(* IEC 61131-3 sources: DemoPumpStation/Testing, 3 files *)

(* ---- test_pdi_codec.st ---- *)
// @Test "PdiCodec decode with both command bits cleared"
// @data (control:=0, powerWord:=0, expectedStart:=0, expectedStop:=0, expectedPower:=0.0)
FUNCTION Test_PdiCodec_Decode_NoCommands : bool
VAR_INPUT
    control : word;
    powerWord : word;
    expectedStart : bool;
    expectedStop : bool;
    expectedPower : real;
END_VAR
VAR
    codec : PdiCodec;
    entry : PumpStationControl;
    words : array[0..1] of word;
    seg : Modbus.ModbusSegment;
END_VAR
    // Arrange
    words[0] := control;
    words[1] := powerWord;
    seg.attachReadable('mbs', Modbus.ModbusArea#holds, 0, ref(words));
    codec.init(0, seg);

    entry.startCmd := true;
    entry.stopCmd := true;
    entry.setpointPower := -999.0;

    // Act
    codec.decode(entry);

    // Assert
    Test_PdiCodec_Decode_NoCommands :=
        (entry.startCmd = expectedStart) and
        (entry.stopCmd = expectedStop) and
        (entry.setpointPower = expectedPower);
END_FUNCTION

// @Test "PdiCodec decode start command only"
// @data (control:=1, powerWord:=100, expectedStart:=1, expectedStop:=0, expectedPower:=100.0)
FUNCTION Test_PdiCodec_Decode_StartOnly : bool
VAR_INPUT
    control : word;
    powerWord : word;
    expectedStart : bool;
    expectedStop : bool;
    expectedPower : real;
END_VAR
VAR
    codec : PdiCodec;
    entry : PumpStationControl;
    words : array[0..1] of word;
    seg : Modbus.ModbusSegment;
END_VAR
    words[0] := control;
    words[1] := powerWord;

    seg.attachReadable('mbs', Modbus.ModbusArea#holds, 0, ref(words));
    codec.init(0, seg);

    entry.startCmd := false;
    entry.stopCmd := true;
    entry.setpointPower := -1.0;

    codec.decode(entry);

    Test_PdiCodec_Decode_StartOnly :=
        (entry.startCmd = expectedStart) and
        (entry.stopCmd = expectedStop) and
        (entry.setpointPower = expectedPower);
END_FUNCTION

// @Test "PdiCodec decode stop command only"
// @data (control:=2, powerWord:=250, expectedStart:=0, expectedStop:=1, expectedPower:=250.0)
FUNCTION Test_PdiCodec_Decode_StopOnly : bool
VAR_INPUT
    control : word;
    powerWord : word;
    expectedStart : bool;
    expectedStop : bool;
    expectedPower : real;
END_VAR
VAR
    codec : PdiCodec;
    entry : PumpStationControl;
    words : array[0..1] of word;
    seg : Modbus.ModbusSegment;
END_VAR
    words[0] := control;
    words[1] := powerWord;
    seg.attachReadable('mbs', Modbus.ModbusArea#holds, 0, ref(words));
    codec.init(0, seg);

    entry.startCmd := true;
    entry.stopCmd := false;
    entry.setpointPower := -1.0;

    codec.decode(entry);

    Test_PdiCodec_Decode_StopOnly :=
        (entry.startCmd = expectedStart) and
        (entry.stopCmd = expectedStop) and
        (entry.setpointPower = expectedPower);
END_FUNCTION

// @Test "PdiCodec decode both command bits set"
// @data (control:=3, powerWord:=500, expectedStart:=1, expectedStop:=1, expectedPower:=500.0)
FUNCTION Test_PdiCodec_Decode_BothCommands : bool
VAR_INPUT
    control : word;
    powerWord : word;
    expectedStart : bool;
    expectedStop : bool;
    expectedPower : real;
END_VAR
VAR
    codec : PdiCodec;
    entry : PumpStationControl;
    words : array[0..1] of word;
    seg : Modbus.ModbusSegment;
END_VAR
    words[0] := control;
    words[1] := powerWord;
    seg.attachReadable('mbs', Modbus.ModbusArea#holds, 0, ref(words));
    codec.init(0, seg);

    entry.startCmd := false;
    entry.stopCmd := false;
    entry.setpointPower := -1.0;

    codec.decode(entry);

    Test_PdiCodec_Decode_BothCommands :=
        (entry.startCmd = expectedStart) and
        (entry.stopCmd = expectedStop) and
        (entry.setpointPower = expectedPower);
END_FUNCTION

// @Test "PdiCodec decode ignores unrelated control bits"
// @data (control:=16#0004, powerWord:=77, expectedStart:=0, expectedStop:=0, expectedPower:=77.0)
// @data (control:=16#8000, powerWord:=88, expectedStart:=0, expectedStop:=0, expectedPower:=88.0)
// @data (control:=16#FFFF, powerWord:=99, expectedStart:=1, expectedStop:=1, expectedPower:=99.0)
FUNCTION Test_PdiCodec_Decode_IgnoreOtherBits : bool
VAR_INPUT
    control : word;
    powerWord : word;
    expectedStart : bool;
    expectedStop : bool;
    expectedPower : real;
END_VAR
VAR
    codec : PdiCodec;
    entry : PumpStationControl;
    words : array[0..1] of word;
    seg : Modbus.ModbusSegment;
END_VAR
    words[0] := control;
    words[1] := powerWord;
    seg.attachReadable('mbs', Modbus.ModbusArea#holds, 0, ref(words));
    codec.init(0, seg);

    entry.startCmd := false;
    entry.stopCmd := false;
    entry.setpointPower := -1.0;

    codec.decode(entry);

    Test_PdiCodec_Decode_IgnoreOtherBits :=
        (entry.startCmd = expectedStart) and
        (entry.stopCmd = expectedStop) and
        (entry.setpointPower = expectedPower);
END_FUNCTION

// @Test "PdiCodec decode from non zero offset"
// @data (dummy0:=111, control:=3, powerWord:=222, expectedStart:=1, expectedStop:=1, expectedPower:=222.0)
FUNCTION Test_PdiCodec_Decode_WithOffset : bool
VAR_INPUT
    dummy0 : word;
    control : word;
    powerWord : word;
    expectedStart : bool;
    expectedStop : bool;
    expectedPower : real;
END_VAR
VAR
    codec : PdiCodec;
    entry : PumpStationControl;
    words : array[0..2] of word;
    seg : Modbus.ModbusSegment;
END_VAR
    words[0] := dummy0;
    words[1] := control;
    words[2] := powerWord;

    seg.attachReadable('mbs', Modbus.ModbusArea#holds, 0, ref(words));
    codec.init(1, seg);

    entry.startCmd := false;
    entry.stopCmd := false;
    entry.setpointPower := -1.0;

    codec.decode(entry);

    Test_PdiCodec_Decode_WithOffset :=
        (entry.startCmd = expectedStart) and
        (entry.stopCmd = expectedStop) and
        (entry.setpointPower = expectedPower);
END_FUNCTION

// @Test "PdiCodec decode advances offset by two words"
FUNCTION Test_PdiCodec_Decode_UpdatesOffset : bool
VAR
    codec : PdiCodec;
    entry : PumpStationControl;
    words : array[0..3] of word;
    seg : Modbus.ModbusSegment;
END_VAR
    words[0] := 3;
    words[1] := 100;
    words[2] := 555;
    words[3] := 777;

    seg.attachReadable('mbs', Modbus.ModbusArea#holds, 0, ref(words));
    codec.init(0, seg);

    codec.decode(entry);

    Test_PdiCodec_Decode_UpdatesOffset := codec.getCurrentOffset() = 2;
END_FUNCTION

(* ---- test_pdo.codec.st ---- *)
// @Test "PdoCodec encode PumpUnitView basic field mapping"
// @data (id:=16#12345678, expectedIdLo:=16#5678, expectedIdHi:=16#1234, role:=7, available:=1, faulted:=0, active:=1, power:=12.3, expectedStates:=5, expectedPower:=123)
FUNCTION Test_PdoCodec_Encode_PumpUnitView_Basic : bool
VAR_INPUT
    id : dword;
    expectedIdLo : word;
    expectedIdHi : word;
    role : PumpRole;
    available : bool;
    faulted : bool;
    active : bool;
    power : real;
    expectedStates : word;
    expectedPower : word;
END_VAR
VAR
    codec : PdoCodec;
    seg : Modbus.ModbusSegment;
    words : array[0..7] of word;
    entry : PumpUnitView;
END_VAR
    // Arrange
    entry.id := id;
    entry.role := role;
    entry.available := available;
    entry.faulted := faulted;
    entry.active := active;
    entry.power := power;

    seg.attachWritable('mbs', Modbus.ModbusArea#inputs, 0, ref(words));
    codec.init(0, seg);

    // Act
    codec.encode(ref(entry));

    // Assert
    Test_PdoCodec_Encode_PumpUnitView_Basic :=
        (words[0] = expectedIdLo) and
        (words[1] = expectedIdHi) and
        (words[2] = role) and
        (words[3] = expectedStates) and
        (words[4] = expectedPower) and
        (codec.getCurrentOffset() = 5);
END_FUNCTION

// @Test "PdoCodec encode PumpUnitView state bit packing"
// @data (available:=0, faulted:=0, active:=0, expectedStates:=0)
// @data (available:=1, faulted:=0, active:=0, expectedStates:=1)
// @data (available:=0, faulted:=1, active:=0, expectedStates:=2)
// @data (available:=0, faulted:=0, active:=1, expectedStates:=4)
// @data (available:=1, faulted:=1, active:=0, expectedStates:=3)
// @data (available:=1, faulted:=0, active:=1, expectedStates:=5)
// @data (available:=0, faulted:=1, active:=1, expectedStates:=6)
// @data (available:=1, faulted:=1, active:=1, expectedStates:=7)
FUNCTION Test_PdoCodec_Encode_PumpUnitView_States : bool
VAR_INPUT
    available : bool;
    faulted : bool;
    active : bool;
    expectedStates : word;
END_VAR
VAR
    codec : PdoCodec;
    seg : Modbus.ModbusSegment;
    words : array[0..7] of word;
    entry : PumpUnitView;
END_VAR
    // Arrange
    words[0] := 16#AAAA;
    words[1] := 16#BBBB;
    words[2] := 16#CCCC;
    words[3] := 16#DDDD;
    words[4] := 16#EEEE;
    words[5] := 16#FFFF;
    words[6] := 16#1111;
    words[7] := 16#2222;

    entry.id := 1;
    entry.role := 2;
    entry.available := available;
    entry.faulted := faulted;
    entry.active := active;
    entry.power := 0.0;

    seg.attachWritable('mbs', Modbus.ModbusArea#inputs, 0, ref(words));
    codec.init(0, seg);

    // Act
    codec.encode(ref(entry));

    // Assert
    Test_PdoCodec_Encode_PumpUnitView_States := words[3] = expectedStates;
END_FUNCTION

// @Test "PdoCodec encode PumpUnitView from non zero offset"
// @data (startOffset:=2, id:=16#00000001, role:=9, available:=1, faulted:=1, active:=0, power:=4.2, expectedStates:=3, expectedPower:=42)
FUNCTION Test_PdoCodec_Encode_PumpUnitView_WithOffset : bool
VAR_INPUT
    startOffset : uint;
    id : dword;
    role : PumpRole;
    available : bool;
    faulted : bool;
    active : bool;
    power : real;
    expectedStates : word;
    expectedPower : word;
END_VAR
VAR
    codec : PdoCodec;
    seg : Modbus.ModbusSegment;
    words : array[0..9] of word;
    entry : PumpUnitView;
END_VAR
    // Arrange
    words[0] := 111;
    words[1] := 222;
    words[2] := 0;
    words[3] := 0;
    words[4] := 0;
    words[5] := 0;
    words[6] := 0;
    words[7] := 0;
    words[8] := 999;
    words[9] := 888;

    entry.id := id;
    entry.role := role;
    entry.available := available;
    entry.faulted := faulted;
    entry.active := active;
    entry.power := power;

    seg.attachWritable('mbs', Modbus.ModbusArea#inputs, 0, ref(words));
    codec.init(startOffset, seg);

    // Act
    codec.encode(ref(entry));

    // Assert
    Test_PdoCodec_Encode_PumpUnitView_WithOffset :=
        (words[startOffset + 2] = role) and
        (words[startOffset + 3] = expectedStates) and
        (words[startOffset + 4] = expectedPower) and
        (codec.getCurrentOffset() = startOffset + 5);
END_FUNCTION

// -@Test "PdoCodec encode PumpControllerViewModel basic field mapping"
// @data (isStarted:=1, vfdStatus:=0, vfdUnitId:=25, requestedPower:=10.0, vfdFrequency:=50.0, activePower:=8.5, expectedStates:=1, expectedRequested:=100, expectedFreq:=500, expectedActive:=85)
FUNCTION Test_PdoCodec_Encode_Controller_Basic : bool
VAR_INPUT
    isStarted : bool;
    vfdStatus : bool;
    vfdUnitId : udint;
    requestedPower : real;
    vfdFrequency : real;
    activePower : real;
    expectedStates : word;
    expectedRequested : word;
    expectedFreq : word;
    expectedActive : word;
END_VAR
VAR
    codec : PdoCodec;
    seg : Modbus.ModbusSegment;
    words : array[0..7] of word;
    entry : PumpControllerViewModel;
END_VAR
    // Arrange
    words[0] := 0;
    words[1] := 0;
    words[2] := 0;
    words[3] := 0;
    words[4] := 0;
    words[5] := 0;
    words[6] := 0;
    words[7] := 0;

    entry.isStarted := isStarted;
    entry.vfdStatus := vfdStatus;
    entry.vfdUnitId := vfdUnitId;
    entry.requestedPower := requestedPower;
    entry.vfdFrequency := vfdFrequency;
    entry.activePower := activePower;

    seg.attachWritable('mbs', Modbus.ModbusArea#inputs, 0, ref(words));
    codec.init(0, seg);

    // Act
    codec.encode(ref(entry));

    // Assert
    Test_PdoCodec_Encode_Controller_Basic :=
        (words[0] = expectedStates) and
        (words[1] = udint_to_word(vfdUnitId)) and
        (words[2] = expectedRequested) and
        (words[3] = expectedFreq) and
        (words[4] = expectedActive) and
        (codec.getCurrentOffset() = 5);
END_FUNCTION

// -@Test "PdoCodec encode PumpControllerViewModel state bit packing"
// @data (isStarted:=0, vfdStatus:=0, expectedStates:=0)
// @data (isStarted:=1, vfdStatus:=0, expectedStates:=1)
// @data (isStarted:=0, vfdStatus:=1, expectedStates:=2)
// @data (isStarted:=1, vfdStatus:=1, expectedStates:=3)
FUNCTION Test_PdoCodec_Encode_Controller_States : bool
VAR_INPUT
    isStarted : bool;
    vfdStatus : bool;
    expectedStates : word;
END_VAR
VAR
    codec : PdoCodec;
    seg : Modbus.ModbusSegment;
    words : array[0..7] of word;
    entry : PumpControllerViewModel;
END_VAR
    // Arrange
    words[0] := 16#FFFF;
    words[1] := 16#FFFF;
    words[2] := 16#FFFF;
    words[3] := 16#FFFF;
    words[4] := 16#FFFF;
    words[5] := 16#FFFF;
    words[6] := 16#FFFF;
    words[7] := 16#FFFF;

    entry.isStarted := isStarted;
    entry.vfdStatus := vfdStatus;
    entry.vfdUnitId := 1;
    entry.requestedPower := 0.0;
    entry.vfdFrequency := 0.0;
    entry.activePower := 0.0;

    seg.attachWritable('mbs', Modbus.ModbusArea#inputs, 0, ref(words));
    codec.init(0, seg);

    // Act
    codec.encode(ref(entry));

    // Assert
    Test_PdoCodec_Encode_Controller_States := words[0] = expectedStates;
END_FUNCTION

// -@Test "PdoCodec encode PumpControllerViewModel from non zero offset"
// @data (startOffset:=3, isStarted:=1, vfdStatus:=1, vfdUnitId:=17, requestedPower:=12.5, vfdFrequency:=48.7, activePower:=11.1, expectedStates:=3, expectedRequested:=125, expectedFreq:=487, expectedActive:=111)
FUNCTION Test_PdoCodec_Encode_Controller_WithOffset : bool
VAR_INPUT
    startOffset : uint;
    isStarted : bool;
    vfdStatus : bool;
    vfdUnitId : udint;
    requestedPower : real;
    vfdFrequency : real;
    activePower : real;
    expectedStates : word;
    expectedRequested : word;
    expectedFreq : word;
    expectedActive : word;
END_VAR
VAR
    codec : PdoCodec;
    seg : Modbus.ModbusSegment;
    words : array[0..11] of word;
    entry : PumpControllerViewModel;
END_VAR
    // Arrange
    words[0] := 101;
    words[1] := 102;
    words[2] := 103;
    words[3] := 0;
    words[4] := 0;
    words[5] := 0;
    words[6] := 0;
    words[7] := 0;
    words[8] := 999;
    words[9] := 998;
    words[10] := 997;
    words[11] := 996;

    entry.isStarted := isStarted;
    entry.vfdStatus := vfdStatus;
    entry.vfdUnitId := vfdUnitId;
    entry.requestedPower := requestedPower;
    entry.vfdFrequency := vfdFrequency;
    entry.activePower := activePower;

    seg.attachWritable('mbs', Modbus.ModbusArea#inputs, 0, ref(words));
    codec.init(startOffset, seg);

    // Act
    codec.encode(ref(entry));

    // Assert
    Test_PdoCodec_Encode_Controller_WithOffset :=
        (words[startOffset + 0] = expectedStates) and
        (words[startOffset + 1] = udint_to_word(vfdUnitId)) and
        (words[startOffset + 2] = expectedRequested) and
        (words[startOffset + 3] = expectedFreq) and
        (words[startOffset + 4] = expectedActive) and
        (codec.getCurrentOffset() = startOffset + 5);
END_FUNCTION

(* ---- test_units_manager.st ---- *)
// @Test "UnitManager init assigns sequential ids and correct size"
FUNCTION Test_UnitManager_Init_SizeAndIds : bool
VAR
    mgr : UnitManager;
    units : array[5..7] of PumpUnit;
END_VAR
    // Act
    mgr.init(ref(units), 10.0);

    // Assert
    Test_UnitManager_Init_SizeAndIds :=
        (units[5].id = 1) and
        (units[6].id = 2) and
        (units[7].id = 3);
END_FUNCTION

// @Test "UnitManager init with null collection keeps manager empty"
FUNCTION Test_UnitManager_Init_NullCollection : bool
VAR
    mgr : UnitManager;
    h : unitHandle;
END_VAR
    // Act
    mgr.init(NULL, 10.0);
    h := mgr.findNextAvailable();

    // Assert
    Test_UnitManager_Init_NullCollection :=
        (h = NULL);
END_FUNCTION

// @Test "UnitManager findUnit returns handle for existing unit id"
FUNCTION Test_UnitManager_FindUnit_Existing : bool
VAR
    mgr : UnitManager;
    units : array[1..3] of PumpUnit;
    h : unitHandle;
END_VAR
    // Arrange
    mgr.init(ref(units), 10.0);

    // Act
    h := mgr.findUnit(2);

    // Assert
    Test_UnitManager_FindUnit_Existing :=
        (h <> NULL) and
        (h^.id = 2);
END_FUNCTION

// @Test "UnitManager findUnit returns null for missing id"
FUNCTION Test_UnitManager_FindUnit_Missing : bool
VAR
    mgr : UnitManager;
    units : array[1..3] of PumpUnit;
    h : unitHandle;
END_VAR
    // Arrange
    mgr.init(ref(units), 10.0);

    // Act
    h := mgr.findUnit(99);

    // Assert
    Test_UnitManager_FindUnit_Missing := h = NULL;
END_FUNCTION

// @Test "UnitManager findNextAvailable returns first available non faulted inactive unit"
FUNCTION Test_UnitManager_FindNextAvailable_FirstMatch : bool
VAR
    mgr : UnitManager;
    units : array[1..4] of PumpUnit;
    h : unitHandle;
END_VAR
    // Arrange
    mgr.init(ref(units), 10.0);

    units[1].available := false;
    units[1].faulted := false;
    units[1].role := PumpRole#stopped;

    units[2].available := true;
    units[2].faulted := true;
    units[2].role := PumpRole#stopped;

    units[3].available := true;
    units[3].faulted := false;
    units[3].role := PumpRole#stopped;

    units[4].available := true;
    units[4].faulted := false;
    units[4].role := PumpRole#stopped;

    // Act
    h := mgr.findNextAvailable();

    // Assert
    Test_UnitManager_FindNextAvailable_FirstMatch :=
        (h <> NULL) and
        (h^.id = 3);
END_FUNCTION

// @Test "UnitManager findNextAvailable skips active units"
// @data (role1:=0, role2:=1, expectedId:=2)
FUNCTION Test_UnitManager_FindNextAvailable_SkipsActive : bool
VAR_INPUT
    role1 : PumpRole;
    role2 : PumpRole;
    expectedId : udint;
END_VAR
VAR
    mgr : UnitManager;
    units : array[1..2] of PumpUnit;
    h : unitHandle;
END_VAR
    // Arrange
    mgr.init(ref(units), 10.0);

    units[1].available := true;
    units[1].faulted := false;
    units[1].role := role1;

    units[2].available := true;
    units[2].faulted := false;
    units[2].role := role2;

    // Act
    h := mgr.findNextAvailable();

    // Assert
    Test_UnitManager_FindNextAvailable_SkipsActive :=
        (h <> NULL) and
        (h^.id = expectedId);
END_FUNCTION

// @Test "UnitManager findNextAvailable returns null when no unit is eligible"
FUNCTION Test_UnitManager_FindNextAvailable_None : bool
VAR
    mgr : UnitManager;
    units : array[1..3] of PumpUnit;
    h : unitHandle;
END_VAR
    // Arrange
    mgr.init(ref(units), 10.0);

    units[1].available := false;
    units[2].available := true;
    units[2].faulted := true;
    units[3].available := true;
    units[3].faulted := false;
    units[3].role := PumpRole#onVfd;

    // Act
    h := mgr.findNextAvailable();

    // Assert
    Test_UnitManager_FindNextAvailable_None := h = NULL;
END_FUNCTION

// @Test "UnitManager findBypassUnit returns first bypass unit"
FUNCTION Test_UnitManager_FindBypassUnit_FirstMatch : bool
VAR
    mgr : UnitManager;
    units : array[1..4] of PumpUnit;
    h : unitHandle;
END_VAR
    // Arrange
    mgr.init(ref(units), 10.0);

    units[1].role := PumpRole#stopped;
    units[2].role := PumpRole#onVfd;
    units[3].role := PumpRole#onBypass;
    units[4].role := PumpRole#onBypass;

    // Act
    h := mgr.findBypassUnit();

    // Assert
    Test_UnitManager_FindBypassUnit_FirstMatch :=
        (h <> NULL) and
        (h^.id = 3);
END_FUNCTION

// @Test "UnitManager findBypassUnit returns null when no bypass unit exists"
FUNCTION Test_UnitManager_FindBypassUnit_None : bool
VAR
    mgr : UnitManager;
    units : array[1..3] of PumpUnit;
    h : unitHandle;
END_VAR
    // Arrange
    mgr.init(ref(units), 10.0);

    units[1].role := PumpRole#stopped;
    units[2].role := PumpRole#stopped;
    units[3].role := PumpRole#onVfd;

    // Act
    h := mgr.findBypassUnit();

    // Assert
    Test_UnitManager_FindBypassUnit_None := h = NULL;
END_FUNCTION

// @Test "UnitManager getActiveCount counts active units correctly"
FUNCTION Test_UnitManager_GetActiveCount : bool
VAR
    mgr : UnitManager;
    units : array[1..4] of PumpUnit;
END_VAR
    // Arrange
    mgr.init(ref(units), 10.0);

    units[1].role := PumpRole#stopped;
    units[2].role := PumpRole#onVfd;
    units[3].role := PumpRole#onBypass;
    units[4].role := PumpRole#stopped;

    // Act / Assert
    Test_UnitManager_GetActiveCount := mgr.getActiveCount() = 2;
END_FUNCTION

// @Test "UnitManager getUnitRole returns role by logical id"
FUNCTION Test_UnitManager_GetUnitRole_ById : bool
VAR
    mgr : UnitManager;
    units : array[5..7] of PumpUnit;
END_VAR
    // Arrange
    mgr.init(ref(units), 10.0);

    units[5].role := PumpRole#stopped;   // id = 1
    units[6].role := PumpRole#onBypass;  // id = 2
    units[7].role := PumpRole#onVfd;     // id = 3

    // Assert
    Test_UnitManager_GetUnitRole_ById :=
        mgr.getUnitRole(2) = PumpRole#onBypass;
END_FUNCTION

// @Test "UnitManager getUnitAvailable returns availability by logical id"
FUNCTION Test_UnitManager_GetUnitAvailable_ById : bool
VAR
    mgr : UnitManager;
    units : array[5..7] of PumpUnit;
END_VAR
    // Arrange
    mgr.init(ref(units), 10.0);

    units[5].available := false; // id = 1
    units[6].available := true;  // id = 2
    units[7].available := false; // id = 3

    // Assert
    Test_UnitManager_GetUnitAvailable_ById := mgr.getUnitAvailable(2);
END_FUNCTION

// @Test "UnitManager getUnitFaulted returns fault state by logical id"
FUNCTION Test_UnitManager_GetUnitFaulted_ById : bool
VAR
    mgr : UnitManager;
    units : array[5..7] of PumpUnit;
END_VAR
    // Arrange
    mgr.init(ref(units), 10.0);

    units[5].faulted := false; // id = 1
    units[6].faulted := true;  // id = 2
    units[7].faulted := false; // id = 3

    // Assert
    Test_UnitManager_GetUnitFaulted_ById := mgr.getUnitFaulted(2);
END_FUNCTION

// @Test "UnitManager getCurrentPower sums performance of all units"
FUNCTION Test_UnitManager_GetCurrentPower_Sum : bool
VAR
    mgr : UnitManager;
    units : array[1..3] of PumpUnit;
    power : real;
END_VAR
    // Arrange
    mgr.init(ref(units), 10.0);

    units[1].role := PumpRole#onVfd;
    units[2].role := PumpRole#onBypass;
    units[3].role := PumpRole#stopped;

    // Act
    power := mgr.getCurrentPower(50.0);

    // Assert
    Test_UnitManager_GetCurrentPower_Sum := power > 0.0;
END_FUNCTION
